//==============================================================
// 单轴外部命令保护
//
// 职责：
// 1. 通信无效时清除指定轴的全部外部命令；
// 2. 锁存通信恢复后的命令复位要求；
// 3. 旧命令全部清零后重新开放控制；
// 4. 不直接调用任何PLCopen运动功能块。
//==============================================================

FUNCTION_BLOCK FB_AxisCommandGuard

VAR_INPUT
    bProtectionEnabled : BOOL;     // 是否启用HMI通信保护
    bCommunicationOnline : BOOL;   // FB_HmiWatchdog输出的在线状态
    bHoldEnableForStop : BOOL;      // 停止期间不得由通信保护提前撤使能
END_VAR

VAR_IN_OUT
    ioCmd : ST_AxisCmd;            // 需要保护的单轴外部命令
END_VAR

VAR_OUTPUT
    bCommandsSafe : BOOL;          // 本周期进入FB时命令是否全部为FALSE
    bControlAllowed : BOOL;        // 提供给FB_AxisControl的最终控制许可
    bRequireEnableReset : BOOL;    // 通信恢复后是否等待旧命令清零
END_VAR

//==============================================================
// 1. 先检查命令状态
//
// 必须在清理前检查，使通信恢复后至少经过一个完整PLC周期，
// 防止清理和重新授权在同一扫描周期内同时完成。
//==============================================================
bCommandsSafe := M_AreCommandsSafe(
    iCmd := ioCmd
);


//==============================================================
// 2. 生成重新授权锁存和最终控制许可
//==============================================================
IF NOT bProtectionEnabled THEN
    bRequireEnableReset := FALSE;
    bControlAllowed := TRUE;
ELSE
    IF NOT bCommunicationOnline THEN
        bRequireEnableReset := TRUE;
    ELSIF bRequireEnableReset AND bCommandsSafe THEN
        bRequireEnableReset := FALSE;
    END_IF;

    bControlAllowed :=
        bCommunicationOnline
        AND NOT bRequireEnableReset;
END_IF;


//==============================================================
// 3. 许可无效时统一清理外部命令
//==============================================================
IF NOT bControlAllowed THEN
    M_ClearCommands(
        ioCmd := ioCmd,
        bHoldEnableForStop := bHoldEnableForStop
    );
END_IF;

METHOD PRIVATE M_AreCommandsSafe : BOOL
VAR_INPUT
    iCmd : ST_AxisCmd;
END_VAR
//==============================================================
// 所有可能导致轴动作的命令都必须已经清零，
// 才允许HMI通信恢复后重新开放控制。
//==============================================================
M_AreCommandsSafe :=
    NOT iCmd.bEnable
    AND NOT iCmd.bReset
    AND NOT iCmd.bHome
    AND NOT iCmd.bStop
    AND NOT iCmd.bMoveAbs
    AND NOT iCmd.bMoveRel
    AND NOT iCmd.bJogPos
    AND NOT iCmd.bJogNeg
    AND NOT iCmd.bTorqueControl;
END_METHOD

METHOD PRIVATE M_ClearCommands
VAR_INPUT
    bHoldEnableForStop : BOOL;
END_VAR
VAR_IN_OUT
    ioCmd : ST_AxisCmd;
END_VAR
//==============================================================
// 通信无效时清除所有控制命令并撤销轴使能
//==============================================================
// 停止管理器先执行MC_Stop；其确认后统一撤使能。
IF NOT bHoldEnableForStop THEN
    ioCmd.bEnable := FALSE;
END_IF;

ioCmd.bReset := FALSE;
ioCmd.bHome := FALSE;
ioCmd.bMoveAbs := FALSE;
ioCmd.bMoveRel := FALSE;

ioCmd.bJogPos := FALSE;
ioCmd.bJogNeg := FALSE;

// 必须补充，防止夹紧轴在HMI失联后继续保持转矩。
ioCmd.bTorqueControl := FALSE;
END_METHOD

END_FUNCTION_BLOCK

(* stored: Version 1.1.0.1, ProductVersion 3.1.4026.18
   POU FB_AxisCommandGuard: Id {7cfd58f3-d9dc-4e70-9f98-d249022d8f85}, SpecialFunc None
   Method M_AreCommandsSafe: Id {14fbffeb-c64f-4cc2-9ea3-29e31b274409}
   Method M_ClearCommands: Id {fa777cdb-175b-4e5f-af64-a332007c3aae} *)
